PROGRAM MAIN
VAR
END_VAR

Call_Std_func();

END_PROGRAM

(* stored: Version 1.1.0.1, ProductVersion 3.1.4024.9
   POU MAIN: Id {a4e332ad-eacf-4f7b-a007-da2ec0f7672c}, SpecialFunc None *)
